(* Logix 5000 project; controller Reto1_SeparatingEstation Emulate 5570 rev 30.12; software revision 30.00 *)

TASK MainTask (continuous, watchdog 500 ms) : MainProgram

MODULES
   Local : Emulate 5570 (ICP 2, rev 30.12)
      I_O : vendor 1 type 0 code 15 (ICP 3, rev 1.1, Output RPI 150 ms)
END_MODULES

VAR_GLOBAL   (* controller tags *)
   Ambas : BOOL;
   Banda3 : BOOL;
   Banda4 : BOOL;
   Bandera1_A : BOOL := 1;
   Bandera1_V : BOOL := 1;
   Bandera2_A : BOOL;
   Bandera2_V : BOOL;
   Diferente : BOOL;
   GD_OUT_0 : BOOL := 1;
   GD_OUT_1 : BOOL := 1;
   GD_OUT_2 : BOOL := 1;
   GD_OUT_3 : BOOL := 1;
   Prioridad : BOOL;
   Pusher_Azul : BOOL;
   Pusher_Verde : BOOL;
   Reset : TIMER;
   Sensor_Azul : BOOL := 1;
   Sensor_paso1 : BOOL;
   Sensor_paso2 : BOOL;
   Sensor_Verde : BOOL;
   start : BOOL;
   Stop : BOOL := 1;
   TimerAmbas : TIMER := (PRE := 11000, ACC := 11018);
   TimerAmbas2 : TIMER := (PRE := 1000);
   TimerAzul : TIMER := (PRE := 2000, EN := 1, DN := 1);
   TimerB1_A : TIMER := (PRE := 4000, ACC := 3027);
   TimerB1_V : TIMER := (PRE := 4000, ACC := 3000);
   TimerB2_A : TIMER := (PRE := 1000, ACC := 1013);
   TimerB2_V : TIMER := (PRE := 1000, ACC := 1016);
   TimerPA : TIMER := (PRE := 4000, ACC := 4012);
   TimerPA2 : TIMER := (PRE := 2000);
   TimerPusherA : TIMER := (PRE := 1000);
   TimerPusherV : TIMER := (PRE := 1000);
   TimerPV : TIMER := (PRE := 4000, ACC := 4000);
   TimerPV2 : TIMER := (PRE := 2000);
   TimerV : TIMER := (PRE := 1500);
   TimerVerde : TIMER := (PRE := 2000, ACC := 2018);
   TimerVoff : TIMER := (PRE := 3000);
END_VAR

PROGRAM MainProgram   (* main routine MainRoutine *)

ROUTINE MainRoutine   (* ladder *)
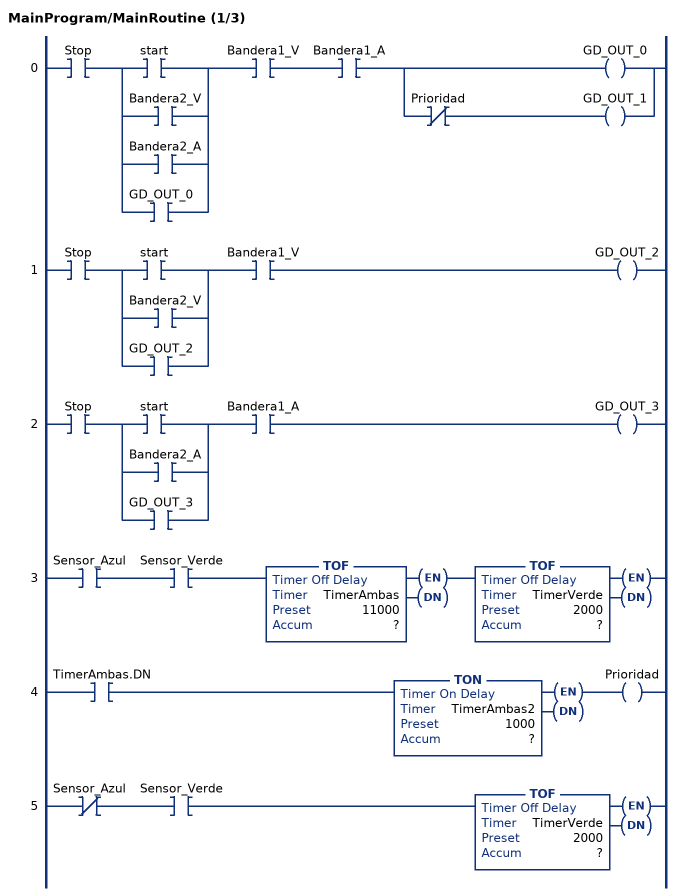
   0: XIC(Stop)[XIC(start) ,XIC(Bandera2_V) ,XIC(Bandera2_A) ,XIC(GD_OUT_0) ]XIC(Bandera1_V)XIC(Bandera1_A)[OTE(GD_OUT_0) ,XIO(Prioridad) OTE(GD_OUT_1) ];
   1: XIC(Stop)[XIC(start) ,XIC(Bandera2_V) ,XIC(GD_OUT_2) ]XIC(Bandera1_V)OTE(GD_OUT_2);
   2: XIC(Stop)[XIC(start) ,XIC(Bandera2_A) ,XIC(GD_OUT_3) ]XIC(Bandera1_A)OTE(GD_OUT_3);
   3: XIC(Sensor_Azul)XIC(Sensor_Verde)TOF(TimerAmbas,?,?)TOF(TimerVerde,?,?);
   4: XIC(TimerAmbas.DN)TON(TimerAmbas2,?,?)OTE(Prioridad);
   5: XIO(Sensor_Azul)XIC(Sensor_Verde)TOF(TimerVerde,?,?);
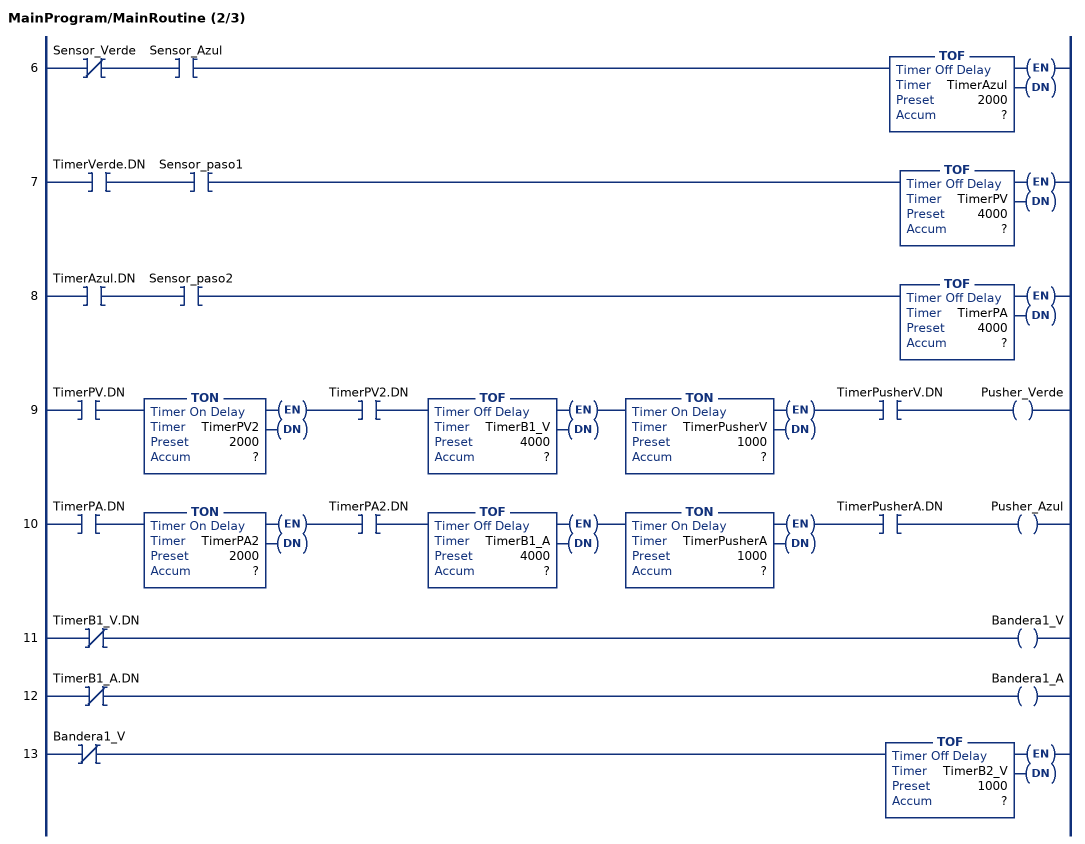
   6: XIO(Sensor_Verde)XIC(Sensor_Azul)TOF(TimerAzul,?,?);
   7: XIC(TimerVerde.DN)XIC(Sensor_paso1)TOF(TimerPV,?,?);
   8: XIC(TimerAzul.DN)XIC(Sensor_paso2)TOF(TimerPA,?,?);
   9: XIC(TimerPV.DN)TON(TimerPV2,?,?)XIC(TimerPV2.DN)TOF(TimerB1_V,?,?)TON(TimerPusherV,?,?)XIC(TimerPusherV.DN)OTE(Pusher_Verde);
   10: XIC(TimerPA.DN)TON(TimerPA2,?,?)XIC(TimerPA2.DN)TOF(TimerB1_A,?,?)TON(TimerPusherA,?,?)XIC(TimerPusherA.DN)OTE(Pusher_Azul);
   11: XIO(TimerB1_V.DN)OTE(Bandera1_V);
   12: XIO(TimerB1_A.DN)OTE(Bandera1_A);
   13: XIO(Bandera1_V)TOF(TimerB2_V,?,?);
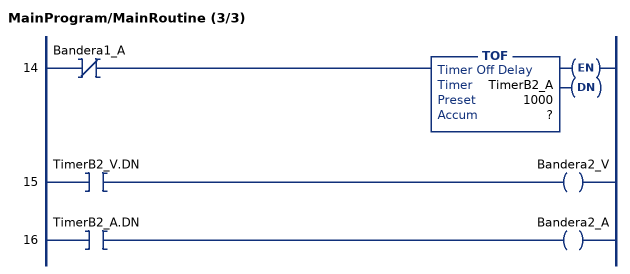
   14: XIO(Bandera1_A)TOF(TimerB2_A,?,?);
   15: XIC(TimerB2_V.DN)OTE(Bandera2_V);
   16: XIC(TimerB2_A.DN)OTE(Bandera2_A);
END_ROUTINE
END_PROGRAM
